TYPE ST_LrParametr :
STRUCT
	lrValue												:	LREAL;
	lrOldValue											:	LREAL;
	lrMinLimit											:	LREAL;
	lrMaxLimit											:	LREAL;
	lrDefault											:	LREAL;
	wsInfoCaption										:	WSTRING(120);	
	wsCaption1											:	WSTRING;
	wsCaption2											:	WSTRING;
	udiColor											:	UDINT	:=	16#FFF0F0F0;	
	bUse2caption										:	BOOL;
	wsUnit												:	WSTRING;
END_STRUCT
END_TYPE

(* stored: Version 1.1.0.1, ProductVersion 3.1.4026.13, FileIdentifier 61edf6fdbf8681d715e480e4479b567bcd128d5b, FileSignature 58b71e32845bada3c126dd4498aea001f0837f56be478506522056d74918b4e7b7487735ff9f6f40d183e605654b8254edb932f727e097d56653f62dc307b26a44bb4cfb21ec26c96dad46b2653e3526a66f1086cd673007b1a9b92a2e8cfdfdce9cbc0d504a9b60397b8c31bba9a2c5d43165cc237ce40124bbef9c1ab4fda740f306e746892b8f735353968bbd801fd512804e5ca8e2f3e24968c610c1e5436de53122bfa695fbcbfe8d6c23b7d4e0b4df071e44b95e198fedcfd978921aab5f8c0ff877f911625bf92368dd8b2da6148e86f185e977868e6b4eccdc43560a4d5257480ac9d406ac6ed76b4b08ed45ee2ab4c50a8288f7c0c66e70fc43c9ec
   DUT ST_LrParametr: Id {bd4fcfec-ffa6-443d-a5b5-f7b1be52d8fa} *)
